PROGRAM MAIN
VAR
END_VAR

END_PROGRAM

(* stored: Version 1.1.0.1
   POU MAIN: Id {b07b1735-c9b8-4c55-b544-402837ba1c9e} *)
